(* IEC 61131-3 sources: RL_MAR/experiments/comparison/autoplc/results/gpt-4o-mini_20260511_164212/med_38, 1 file *)

(* ---- med_38_1.st ---- *)
FUNCTION_BLOCK SolarPanelTracking
VAR_INPUT
    SolarIntensity : REAL;      (* Input: Solar intensity in percentage *)
    CurrentTime : TIME;         (* Input: Current time of day *)
END_VAR

VAR_OUTPUT
    PanelAngle : REAL := 0.0;   (* Output: Panel angle in degrees *)
END_VAR

VAR
    SunriseTime : TIME := T#6H;    (* Sunrise time set to 6 AM *)
    SunsetTime : TIME := T#18H;     (* Sunset time set to 6 PM *)
    NoonTime : TIME := T#12H;       (* Noon time set to 12 PM *)
    MorningAngle : REAL := 30.0;     (* Angle during morning *)
    NoonAngle : REAL := 60.0;        (* Angle during noon *)
    EveningAngle : REAL := 30.0;      (* Angle during evening *)
END_VAR

(* Main control logic *)
IF CurrentTime < SunriseTime OR CurrentTime > SunsetTime THEN
    PanelAngle := 0.0; (* Nighttime State *)
ELSE
    IF CurrentTime >= SunriseTime AND CurrentTime < NoonTime THEN
        PanelAngle := MorningAngle; (* Morning State *)
    ELSIF CurrentTime = NoonTime THEN
        PanelAngle := NoonAngle; (* Noon State *)
    ELSIF CurrentTime > NoonTime AND CurrentTime < SunsetTime THEN
        IF SolarIntensity >= 90.0 THEN
            PanelAngle := NoonAngle; (* High Solar Intensity State *)
        ELSE
            PanelAngle := EveningAngle; (* Afternoon State *)
        END_IF;
    END_IF;
END_IF;

(* Ensure PanelAngle is within 0 to 90 degrees *)
IF PanelAngle < 0.0 THEN
    PanelAngle := 0.0;
ELSIF PanelAngle > 90.0 THEN
    PanelAngle := 90.0;
END_IF;

END_FUNCTION_BLOCK
